(* CODESYS project gantry3.project

Project tree, tasks and I/O mapping:
  Device : CODESYS Control Win V3, 3S - Smart Software Solutions GmbH, order no. 305021, version 3.5.7.0
    application Application
      libraries: Standard, * (System)
      task MainTask (cyclic, interval t#20ms, priority 1) calls PLC_PRG
      task VISU_TASK (cyclic, interval 100 ms, priority 31) calls VisuElems.Visu_Prg
      program PLC_PRG [LD]
      visualisation Visualization
  text list GlobalTextList
*)

// Device/Application/PLC_PRG
PROGRAM PLC_PRG
VAR
	Step_1: BOOL;
	Start_Btn: BOOL;
	LS_Z_Up: BOOL;
	LS_Y_Home: BOOL;
	LS_X_Home: BOOL;
	Z_Cyl_Down: BOOL;
	LS_Z_Down_Conv: BOOL;
	Step_2: BOOL;
	Vacuum_Valve: BOOL;
	Vac_Sensor: BOOL;
	Step_3: BOOL;
	Step_4: BOOL;
	Y_Cyl_Fwd: BOOL;
	LS_Y_Fwd: BOOL;
	Step_5: BOOL;
	X_Cyl_Fwd: BOOL;
	LS_X_Fwd: BOOL;
	Step_6: BOOL;
	LS_Z_Down_Crate: BOOL;
	Step_7: BOOL;
	Step_8: BOOL;
END_VAR
VAR // added by the converter: edge detectors and wires of the graphical bodies
    _w1, _w2, _w3, _w4, _w5, _w6, _w7 : BOOL;
END_VAR

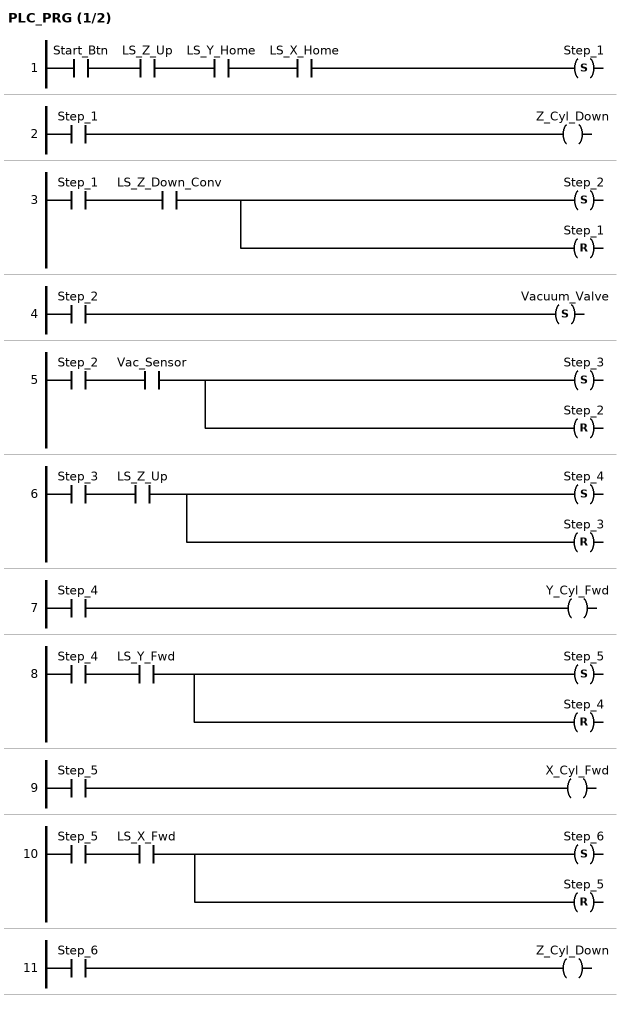
// NETWORK 1
Step_1 S= Start_Btn AND LS_Z_Up AND LS_Y_Home AND LS_X_Home;

// NETWORK 2
Z_Cyl_Down := Step_1;

// NETWORK 3
_w1 := Step_1 AND LS_Z_Down_Conv;
Step_2 S= _w1;
Step_1 R= _w1;

// NETWORK 4
Vacuum_Valve S= Step_2;

// NETWORK 5
_w2 := Step_2 AND Vac_Sensor;
Step_3 S= _w2;
Step_2 R= _w2;

// NETWORK 6
_w3 := Step_3 AND LS_Z_Up;
Step_4 S= _w3;
Step_3 R= _w3;

// NETWORK 7
Y_Cyl_Fwd := Step_4;

// NETWORK 8
_w4 := Step_4 AND LS_Y_Fwd;
Step_5 S= _w4;
Step_4 R= _w4;

// NETWORK 9
X_Cyl_Fwd := Step_5;

// NETWORK 10
_w5 := Step_5 AND LS_X_Fwd;
Step_6 S= _w5;
Step_5 R= _w5;

// NETWORK 11
Z_Cyl_Down := Step_6;

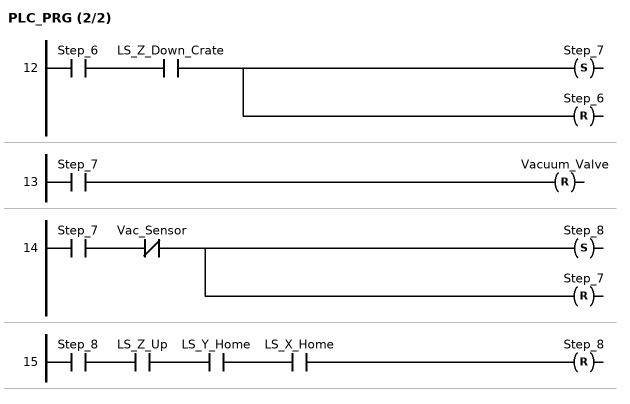
// NETWORK 12
_w6 := Step_6 AND LS_Z_Down_Crate;
Step_7 S= _w6;
Step_6 R= _w6;

// NETWORK 13
Vacuum_Valve R= Step_7;

// NETWORK 14
_w7 := Step_7 AND NOT Vac_Sensor;
Step_8 S= _w7;
Step_7 R= _w7;

// NETWORK 15
Step_8 R= Step_8 AND LS_Z_Up AND LS_Y_Home AND LS_X_Home;

END_PROGRAM

// Device/Application/Visualization
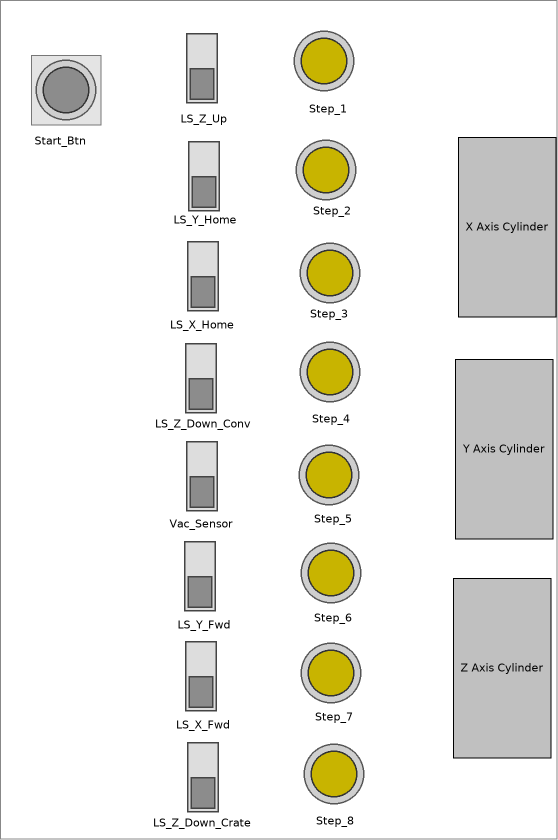
VISUALIZATION Visualization  // 558x840
    PushSwitchLed (31,55 70x70), variable: PLC_PRG.Start_Btn, behaviour: TOGGLE, style: Switch-PushSwitchLed-Gray
    Lamp1 (289,26 70x70), variable: PLC_PRG.Step_1, style: Lamp-Lamp1-Yellow
    Lamp1 (299,739 70x70), variable: PLC_PRG.Step_8, style: Lamp-Lamp1-Yellow
    Lamp1 (296,638 70x70), variable: PLC_PRG.Step_7, style: Lamp-Lamp1-Yellow
    Lamp1 (296,538 70x70), variable: PLC_PRG.Step_6, style: Lamp-Lamp1-Yellow
    Lamp1 (294,440 70x70), variable: PLC_PRG.Step_5, style: Lamp-Lamp1-Yellow
    Lamp1 (291,135 70x70), variable: PLC_PRG.Step_2, style: Lamp-Lamp1-Yellow
    Lamp1 (295,238 70x70), variable: PLC_PRG.Step_3, style: Lamp-Lamp1-Yellow
    Lamp1 (295,337 70x70), variable: PLC_PRG.Step_4, style: Lamp-Lamp1-Yellow
    DipSwitch (169,141 70x70), variable: PLC_PRG.LS_Y_Home, behaviour: TOGGLE, style: Switch-DipSwitch-Gray
    DipSwitch (168,241 70x70), variable: PLC_PRG.LS_X_Home, behaviour: TOGGLE, style: Switch-DipSwitch-Gray
    DipSwitch (166,343 70x70), variable: PLC_PRG.LS_Z_Down_Conv, behaviour: TOGGLE, style: Switch-DipSwitch-Gray
    DipSwitch (167,441 70x70), variable: PLC_PRG.Vac_Sensor, behaviour: TOGGLE, style: Switch-DipSwitch-Gray
    DipSwitch (165,541 70x70), variable: PLC_PRG.LS_Y_Fwd, behaviour: TOGGLE, style: Switch-DipSwitch-Gray
    DipSwitch (166,641 70x70), variable: PLC_PRG.LS_X_Fwd, behaviour: TOGGLE, style: Switch-DipSwitch-Gray
    DipSwitch (168,742 70x70), variable: PLC_PRG.LS_Z_Down_Crate, behaviour: TOGGLE, style: Switch-DipSwitch-Gray
    DipSwitch (167,33 70x70), variable: PLC_PRG.LS_Z_Up, behaviour: TOGGLE, style: Switch-DipSwitch-Gray
    Rectangle (458,137 98x180), "X Axis Cylinder", colour toggle: PLC_PRG.X_Cyl_Fwd
    Rectangle (455,359 98x180), "Y Axis Cylinder", colour toggle: PLC_PRG.Y_Cyl_Fwd
    Rectangle (453,578 98x180), "Z Axis Cylinder", colour toggle: PLC_PRG.Z_Cyl_Down
    Label (10,124 101x34), "Start_Btn"
    Label (129,104 150x30), "LS_Z_Up"
    Label (130,205 150x30), "LS_Y_Home"
    Label (127,310 150x30), "LS_X_Home"
    Label (128,409 150x30), "LS_Z_Down_Conv"
    Label (126,509 150x30), "Vac_Sensor"
    Label (129,610 150x30), "LS_Y_Fwd"
    Label (128,710 150x30), "LS_X_Fwd"
    Label (127,808 150x30), "LS_Z_Down_Crate"
    Label (253,94 150x30), "Step_1"
    Label (260,806 150x30), "Step_8"
    Label (259,702 150x30), "Step_7"
    Label (258,603 150x30), "Step_6"
    Label (258,504 150x30), "Step_5"
    Label (256,404 150x30), "Step_4"
    Label (254,299 150x30), "Step_3"
    Label (257,196 150x30), "Step_2"
END_VISUALIZATION
